TYPE EL2008 :
STRUCT
	Channel_1 AT %Q* : BOOL;
	Channel_2 AT %Q* : BOOL;
	Channel_3 AT %Q* : BOOL;
	Channel_4 AT %Q* : BOOL;
	Channel_5 AT %Q* : BOOL;
	Channel_6 AT %Q* : BOOL;
	Channel_7 AT %Q* : BOOL;
	Channel_8 AT %Q* : BOOL;
END_STRUCT
END_TYPE

(* stored: Version 1.1.0.1, ProductVersion 3.1.4026.18
   DUT EL2008: Id {a8fb9a9a-5645-4e21-bef6-2f5b45345b29} *)
